// Mitsubishi GX Works2 project: 0625(타이머,순차점등2)   PLC: Q02/Q02H

PROGRAM MAIN
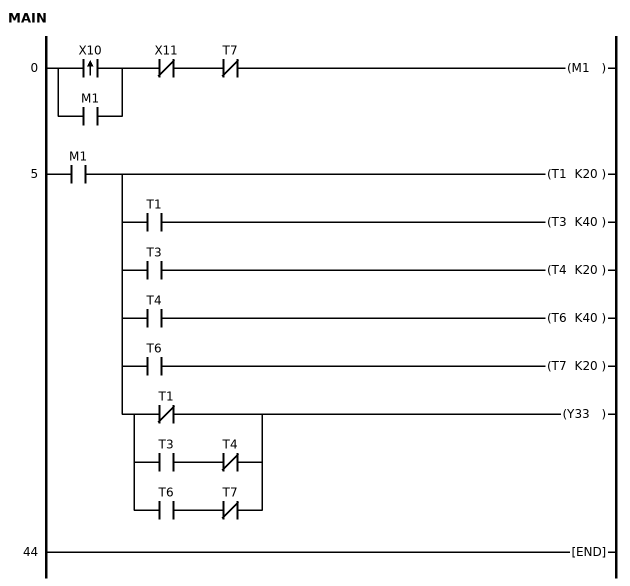
0     LDP     X10
      OR      M1
      ANI     X11
      ANI     T7
      OUT     M1
5     LD      M1
      OUT     T1 K20
      MPS
      AND     T1
      OUT     T3 K40
      MRD
      AND     T3
      OUT     T4 K20
      MRD
      AND     T4
      OUT     T6 K40
      MRD
      AND     T6
      OUT     T7 K20
      MPP
      LDI     T1
      LD      T3
      ANI     T4
      ORB
      LD      T6
      ANI     T7
      ORB
      ANB
      OUT     Y33
44    END
END_PROGRAM
